INTERFACE I_InterfaceManager

METHOD register_I_AI_Percentage : BOOL
VAR_INPUT
	interface_to_be_registered		: I_AI_Percentage;
	terminal_name 					: STRING;
	channel_number 					: USINT; 
END_VAR
VAR_OUTPUT
	errId		: HAL_ErrorEnum;
END_VAR
END_METHOD

METHOD register_I_AI_Voltage : BOOL
VAR_INPUT
	interface_to_be_registered		: I_AI_Voltage;
	terminal_name 					: STRING;
	channel_number 					: USINT; 
END_VAR
VAR_OUTPUT
	errId		: HAL_ErrorEnum;
END_VAR
END_METHOD

METHOD register_terminal : BOOL
VAR_INPUT
	terminal_name : STRING;
END_VAR
VAR_OUTPUT
	errId : HAL_ErrorEnum;
END_VAR
END_METHOD

END_INTERFACE

(* stored: Version 1.1.0.1, ProductVersion 3.1.4024.6
   Itf I_InterfaceManager: Id {bf3d7090-2db7-020e-0254-b2be8a58f566}
   Method register_I_AI_Percentage: Id {7c1c0fdc-f79f-071e-3ef6-8d21c118dda6}
   Method register_I_AI_Voltage: Id {ff6d860c-40ea-058f-1b45-45b6e01389e4}
   Method register_terminal: Id {ff771fff-318e-0cec-18eb-a3ebd10d2480} *)
